ABB RobotStudio station: Desarrollo_RS_20220127-112710.rsstn

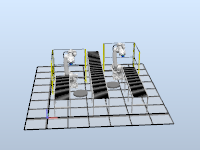
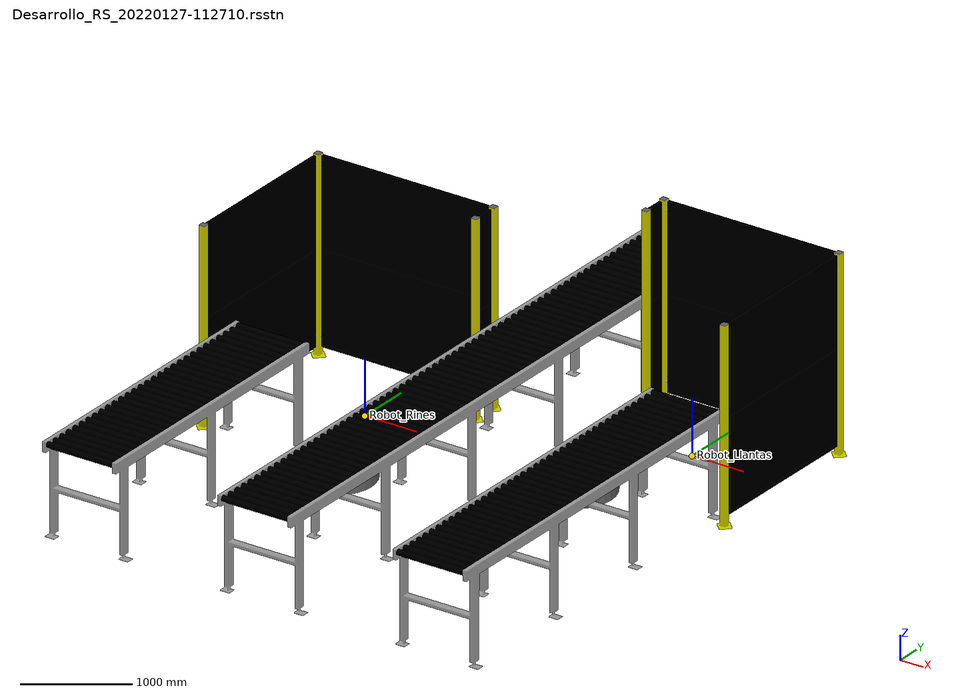
[picture v1: parts stored in the station drawn from their meshes, with robot base, taught points and paths (robot models come from the ABB library and are not in the file)]
Station Station (saved by RobotStudio 21.4.9700.0)
Controller ControladorRobotLlantas, task T_ROB1: task frame (RAPID world) sits at (4075, 4750, 0) mm, rotated rx 0 ry 0 rz -90 deg in the station
Controller ControladorRobotRines, task T_ROB1: task frame (RAPID world) sits at (1225, 3750, 0) mm, rotated rx 0 ry 0 rz -90 deg in the station
Controller ControladorRobotRines
  mechanical unit ROB_1: Robot_Rines, 6 joints, base frame (0, 0, 0) mm
Controller ControladorRobotLlantas
  mechanical unit ROB_1: Robot_Llantas, 6 joints, base frame (0, 0, 0) mm
Layout (positions relative to the parent item):
  - Robot_Rines [mechanism, from Robots\IRB6700_200_260__04.rslib] at (1225, 3750, 0) mm, rotated rx 0 ry 0 rz -90 deg; joint values [0, 0, 0, 0, 0.5236, 0] (rad or m)
  - Robot_Llantas [mechanism, from Robots\IRB6700_200_260__04.rslib] at (4075, 4750, 0) mm, rotated rx 0 ry 0 rz -90 deg; joint values [0, 0, 0, 0, 0.5236, 0] (rad or m)
  - Banda_Rines [part], size 900 x 3000 x 1000 mm
  - Banda_Central [part], size 900 x 7000 x 1000 mm
  - Banda_Llantas [part], size 900 x 4000 x 1000 mm
  - Base_Cepillo_Rines [part], size 800 x 795.6 x 100 mm
  - Base_Cepillo_Llantas [part], size 800 x 795.6 x 100 mm
  - Protector_Robot_Rines [graphiccomponentgroup]
    - Segment 1 [part], size 169.7 x 169.7 x 2000 mm
    - Segment 2 [part], size 169.7 x 359.9 x 2000 mm
    - Segment 3 [part], size 1984.9 x 169.7 x 2000 mm
    - Segment 4 [part], size 169.7 x 1859.9 x 2000 mm
  - Protector_Robot_Llantas [graphiccomponentgroup]
    - Segment 1 [part], size 169.7 x 169.7 x 2000 mm
    - Segment 2 [part], size 169.7 x 359.9 x 2000 mm
    - Segment 3 [part], size 1984.9 x 169.7 x 2000 mm
    - Segment 4 [part], size 169.7 x 1859.9 x 2000 mm
